TYPE E_ConnectionSteps :
(
	eCONNECTION_STATE_IDLE,
	eCONNECTION_STATE_CONNECT_START,
	eCONNECTION_STATE_CONNECT_WAIT,
	eCONNECTION_STATE_DATAEXCHANGE,
	eCONNECTION_STATE_CLOSE_START,
	eCONNECTION_STATE_CLOSE_WAIT,
	eCONNECTION_STATE_ERROR
);
END_TYPE

(* stored: Version 1.1.0.1, ProductVersion 3.1.4024.12
   DUT E_ConnectionSteps: Id {ae46553d-d518-455f-bf7c-ba62e3c0307f} *)
